// TIA Portal V19 export
FUNCTION "EstopStationDecoder" : Void   // FC1, LAD
{ S7_Optimized_Access := 'TRUE' }
// stored: SetENOAutomatically false
   VAR_INPUT
      GreenProcessLamp : Bool;
      BluePushButtonLamp : Bool;
      SelectorSwitchLamp : Bool;
      RedPushButtonLamp : Bool;
      GreenProcessLamp_Raw : Byte;
      BluePushButton_Raw : Byte;
      SelectorSwitch_Raw : Byte;
      RedPushButton_Raw : Byte;
   END_VAR
   VAR_OUTPUT
      GreenProcessActive : Bool;
      BluePushButton : Bool;
      SelectorSwitch : Bool;
      RedPushButton : Bool;
      GreenProcessLamp_Raw_1 : Byte;
      BluePushButtonLamp_Raw : Byte;
      SelectorSwitchLamp_Raw : Byte;
      RedPushButtonLamp_Raw : Byte;
   END_VAR
BEGIN

REGION Network 1: Profinet Estop Decoder
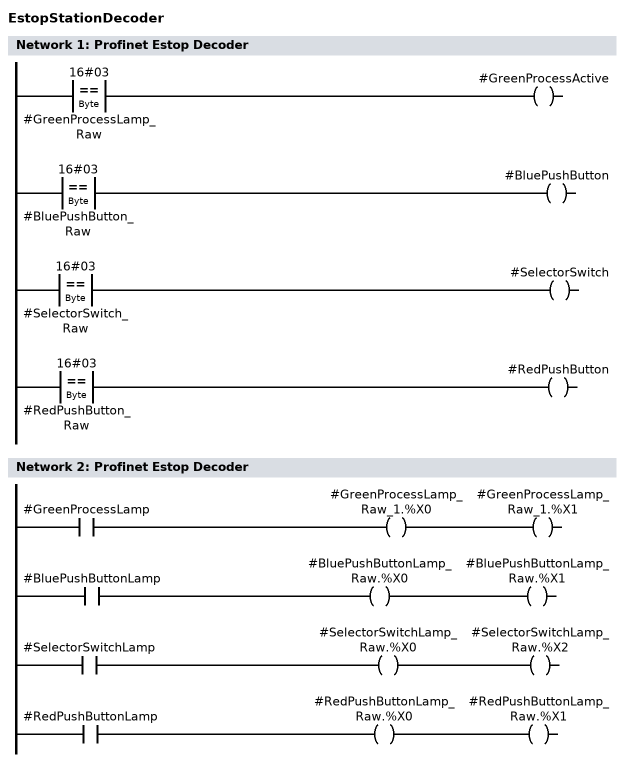
   RUNG wire#powerrail
      { S7_Templates := "SrcType := Byte" } EQ_Contact(in1 := 16#03, in2 := #GreenProcessLamp_Raw)
      Coil( #GreenProcessActive )
   END_RUNG
   RUNG wire#powerrail
      { S7_Templates := "SrcType := Byte" } EQ_Contact(in1 := 16#03, in2 := #BluePushButton_Raw)
      Coil( #BluePushButton )
   END_RUNG
   RUNG wire#powerrail
      { S7_Templates := "SrcType := Byte" } EQ_Contact(in1 := 16#03, in2 := #SelectorSwitch_Raw)
      Coil( #SelectorSwitch )
   END_RUNG
   RUNG wire#powerrail
      { S7_Templates := "SrcType := Byte" } EQ_Contact(in1 := 16#03, in2 := #RedPushButton_Raw)
      Coil( #RedPushButton )
   END_RUNG
   // the same network as SCL:
   #GreenProcessActive := 16#03 = #GreenProcessLamp_Raw;
   #BluePushButton := 16#03 = #BluePushButton_Raw;
   #SelectorSwitch := 16#03 = #SelectorSwitch_Raw;
   #RedPushButton := 16#03 = #RedPushButton_Raw;
END_REGION

REGION Network 2: Profinet Estop Decoder
   RUNG wire#powerrail
      Contact( #GreenProcessLamp )
      Coil( #GreenProcessLamp_Raw_1.%X0 )
      Coil( #GreenProcessLamp_Raw_1.%X1 )
   END_RUNG
   RUNG wire#powerrail
      Contact( #BluePushButtonLamp )
      Coil( #BluePushButtonLamp_Raw.%X0 )
      Coil( #BluePushButtonLamp_Raw.%X1 )
   END_RUNG
   RUNG wire#powerrail
      Contact( #SelectorSwitchLamp )
      Coil( #SelectorSwitchLamp_Raw.%X0 )
      Coil( #SelectorSwitchLamp_Raw.%X2 )
   END_RUNG
   RUNG wire#powerrail
      Contact( #RedPushButtonLamp )
      Coil( #RedPushButtonLamp_Raw.%X0 )
      Coil( #RedPushButtonLamp_Raw.%X1 )
   END_RUNG
   // the same network as SCL:
   #GreenProcessLamp_Raw_1.%X0 := #GreenProcessLamp;
   #GreenProcessLamp_Raw_1.%X1 := #GreenProcessLamp;
   #BluePushButtonLamp_Raw.%X0 := #BluePushButtonLamp;
   #BluePushButtonLamp_Raw.%X1 := #BluePushButtonLamp;
   #SelectorSwitchLamp_Raw.%X0 := #SelectorSwitchLamp;
   #SelectorSwitchLamp_Raw.%X2 := #SelectorSwitchLamp;
   #RedPushButtonLamp_Raw.%X0 := #RedPushButtonLamp;
   #RedPushButtonLamp_Raw.%X1 := #RedPushButtonLamp;
END_REGION
END_FUNCTION
